// TIA Portal V21 export
DATA_BLOCK "PosSenzaDeadBand_DB"   // DB10
// stored: InstanceOfName PosSenzaDeadBand, InstanceOfType FB
"PosSenzaDeadBand"
   // VAR_INPUT
   //    PosRichiesta : Real := 0.0;
   //    PosAttuale : Real := 0.0;
   //    ForzaPos : Bool := FALSE;
   //    ForzaNeg : Bool := FALSE;
   // END_VAR
   // VAR_OUTPUT
   //    Pos : Bool := FALSE;
   //    Neg : Bool := FALSE;
   // END_VAR
   // VAR
   //    DirezioneAvanti : Bool := FALSE;
   //    DirezioneIndietro : Bool := FALSE;
   //    OldPos : Real := 0.0;
   // END_VAR
BEGIN
END_DATA_BLOCK
